Fanuc KAREL source: kb00024.KL

-- PROVISIONAL review KL for V770-1; original PC SHA256 6b72b2a4c1ea5487f355ca17d2a5c62476c638e677a038dfd128f14b8c74a174
-- Incomplete behavior may be omitted. Consult companion uncertainty JSON. Do not deploy.
PROGRAM KB00024
%NOLOCKGROUP
BEGIN
  -- UNRESOLVED_PC offsets 5-15; opcodes 27,22,31
  -- UNRESOLVED_PC offsets 20-24; opcodes 7F
END KB00024
